// TIA Portal V17 export
// export: Created 2025-03-10T12:18:23.2185831Z, ExportSetting WithDefaults, DisplayName Totally Integrated Automation Portal, DisplayVersion V17 Update 8, DisplayName TIA Portal Openness, DisplayVersion V17 Update 8, DisplayName TIA Portal Version Control Interface, DisplayVersion V17, DisplayName SINAMICS Startdrive Advanced, DisplayVersion V17 SP2, DisplayName SINAMICS Startdrive G110M, G120, G120C, G120D, G120P, G115D, DisplayVersion V17 SP2, DisplayName SINAMICS Startdrive G130, G150, S120, S150, SINAMICS MV, S210, DisplayVersion V17 SP2, DisplayName STEP 7 Professional, DisplayVersion V17 Update 8, DisplayName SINUMERIK ONE STEP 7 Toolbox, DisplayVersion V17 Update 12, DisplayName SINUMERIK 840D sl STEP 7 Toolbox, DisplayVersion V17 Update 12, DisplayName STEP 7 Safety, DisplayVersion V17 Update 6, DisplayName WinCC Advanced, DisplayVersion V17 Update 8
ORGANIZATION_BLOCK "OB1_CYCLE"   // OB1, LAD, ProgramCycle
TITLE = "Main Program Sweep (Cycle)"
{ S7_Optimized_Access := 'FALSE' }
VERSION : 0.1
// stored: AutoNumber false, IsIECCheckEnabled false, SetENOAutomatically false
   VAR_TEMP
      EV_CLASS : Byte;   // Bits 0-3 = 1:Coming event, Bits 4-7 = 1:Event class 1
      SCAN_1 : Byte;   // 1:Initial call of the OB, 3: Call 2-n of the OB
      PRIORITY : Byte;   // Priority of OB Execution
      OB_NUMBR : Byte;   // OB number
      RESERVED_1 : Byte;   // Reserved for system
      RESERVED_2 : Byte;   // Reserved for system
      PREV_CYCLE : Int;   // Previous program cycle time (milliseconds)
      MIN_CYCLE : Int;   // Minimum program cycle time (milliseconds)
      MAX_CYCLE : Int;   // Maximum program cycle time (milliseconds)
      DATE_TIME : Date_And_Time;   // Date and time OB started
      OB1_SCAN : Byte;   // 1 (Cold restart scan 1 of OB 1), 3 (Scan 2-n of OB 1)
      OB1_PRIORITY : Int;   // Priority of OB Execution
      OB1_MIN_CYCLE : DInt;   // Minimum cycle time of OB1 (milliseconds)
      OB1_MAX_CYCLE : DInt;   // Maximum cycle time of OB1 (milliseconds)
      PART_TYPE : Int;
      zero : Byte;
      status_sfc21 : Int;
      Error : Bool;
      status : Word;
   END_VAR
   VAR_TEMP   // added for the SCL form of the ladder/FBD networks
      _w1 : Bool;
   END_VAR
BEGIN

REGION Network 1: M ZERO - M ONE
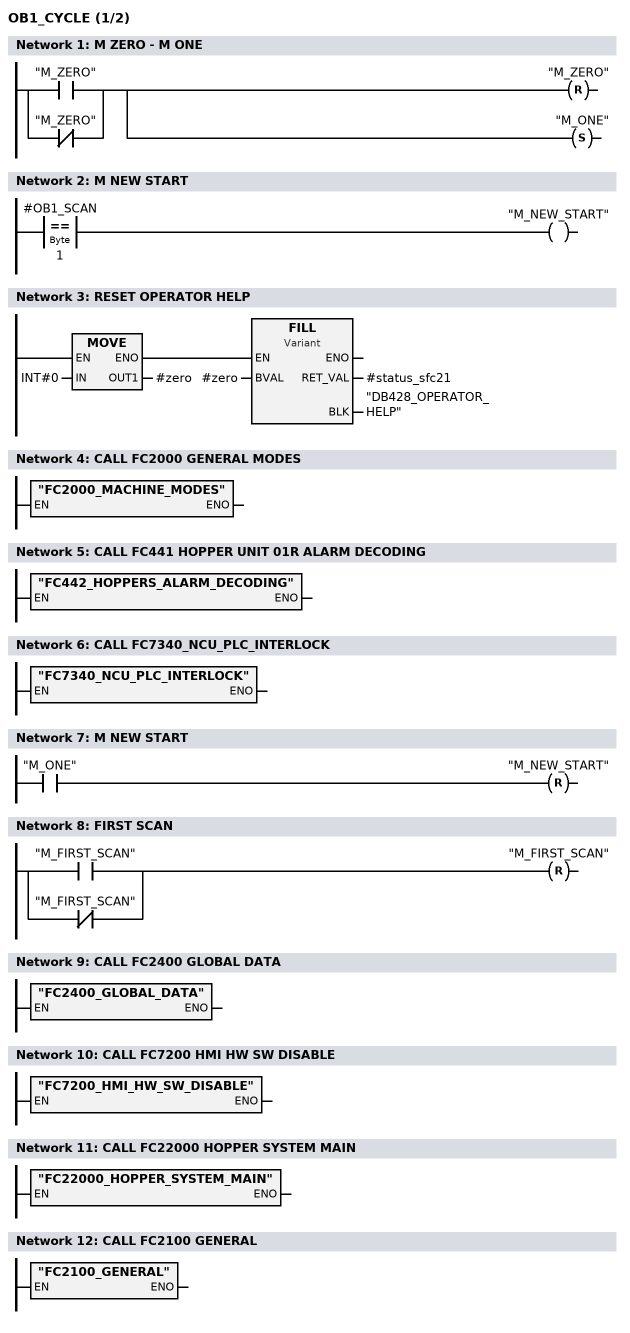
   RUNG wire#powerrail
      Contact( "M_ZERO" )
      wire#w1
      R_Coil( "M_ZERO" )
   END_RUNG
   RUNG wire#powerrail
      I_Contact( "M_ZERO" )
   END_RUNG wire#w1
   RUNG wire#w1
      S_Coil( "M_ONE" )
   END_RUNG
   // the same network as SCL:
   #_w1 := "M_ZERO" OR NOT "M_ZERO";
   IF #_w1 THEN
       "M_ZERO" := FALSE;
       "M_ONE" := TRUE;
   END_IF;
END_REGION

REGION Network 2: M NEW START
   RUNG wire#powerrail
      { S7_Templates := "SrcType := Byte" } EQ_Contact(in1 := #OB1_SCAN, in2 := 1)
      Coil( "M_NEW_START" )
   END_RUNG
   // the same network as SCL:
   "M_NEW_START" := #OB1_SCAN = 1;
END_REGION

REGION Network 3: RESET OPERATOR HELP
   RUNG wire#powerrail
      { S7_GenerateENO := "TRUE" } Move(in := INT#0, out1 => #zero)
      { S7_Templates := "ptr_type := Variant" } FILL(BVAL := #zero, RET_VAL => #status_sfc21, BLK => "DB428_OPERATOR_HELP")
   END_RUNG
   // the same network as SCL:
   // ENO of a box is taken as its EN; it also drops when the box reports an error
   #zero := INT#0;
   #status_sfc21 := FILL(BVAL := #zero, BLK => "DB428_OPERATOR_HELP");
END_REGION

REGION Network 4: CALL FC2000 GENERAL MODES
   RUNG wire#powerrail
      "FC2000_MACHINE_MODES"()
   END_RUNG
   // the same network as SCL:
   "FC2000_MACHINE_MODES"();
END_REGION

REGION Network 5: CALL FC441 HOPPER UNIT 01R ALARM DECODING
   RUNG wire#powerrail
      "FC442_HOPPERS_ALARM_DECODING"()
   END_RUNG
   // the same network as SCL:
   "FC442_HOPPERS_ALARM_DECODING"();
END_REGION

REGION Network 6: CALL FC7340_NCU_PLC_INTERLOCK
   RUNG wire#powerrail
      "FC7340_NCU_PLC_INTERLOCK"()
   END_RUNG
   // the same network as SCL:
   "FC7340_NCU_PLC_INTERLOCK"();
END_REGION

REGION Network 7: M NEW START
   RUNG wire#powerrail
      Contact( "M_ONE" )
      R_Coil( "M_NEW_START" )
   END_RUNG
   // the same network as SCL:
   IF "M_ONE" THEN "M_NEW_START" := FALSE; END_IF;
END_REGION

REGION Network 8: FIRST SCAN
   RUNG wire#powerrail
      Contact( "M_FIRST_SCAN" )
      wire#w1
      R_Coil( "M_FIRST_SCAN" )
   END_RUNG
   RUNG wire#powerrail
      I_Contact( "M_FIRST_SCAN" )
   END_RUNG wire#w1
   // the same network as SCL:
   IF "M_FIRST_SCAN" OR NOT "M_FIRST_SCAN" THEN "M_FIRST_SCAN" := FALSE; END_IF;
END_REGION

REGION Network 9: CALL FC2400 GLOBAL DATA
   RUNG wire#powerrail
      "FC2400_GLOBAL_DATA"()
   END_RUNG
   // the same network as SCL:
   "FC2400_GLOBAL_DATA"();
END_REGION

REGION Network 10: CALL FC7200 HMI HW SW DISABLE
   RUNG wire#powerrail
      "FC7200_HMI_HW_SW_DISABLE"()
   END_RUNG
   // the same network as SCL:
   "FC7200_HMI_HW_SW_DISABLE"();
END_REGION

REGION Network 11: CALL FC22000 HOPPER SYSTEM MAIN
   RUNG wire#powerrail
      "FC22000_HOPPER_SYSTEM_MAIN"()
   END_RUNG
   // the same network as SCL:
   "FC22000_HOPPER_SYSTEM_MAIN"();
END_REGION

REGION Network 12: CALL FC2100 GENERAL
   RUNG wire#powerrail
      "FC2100_GENERAL"()
   END_RUNG
   // the same network as SCL:
   "FC2100_GENERAL"();
END_REGION

REGION Network 13: CALL FC21000 POWDER FEEDER MAIN
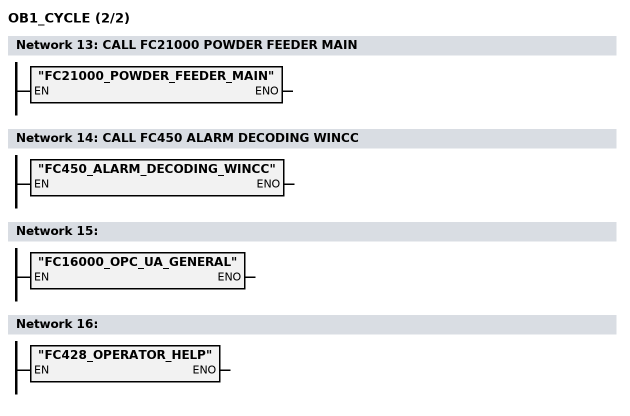
   RUNG wire#powerrail
      "FC21000_POWDER_FEEDER_MAIN"()
   END_RUNG
   // the same network as SCL:
   "FC21000_POWDER_FEEDER_MAIN"();
END_REGION

REGION Network 14: CALL FC450 ALARM DECODING WINCC
   RUNG wire#powerrail
      "FC450_ALARM_DECODING_WINCC"()
   END_RUNG
   // the same network as SCL:
   "FC450_ALARM_DECODING_WINCC"();
END_REGION

REGION Network 15
   RUNG wire#powerrail
      "FC16000_OPC_UA_GENERAL"()
   END_RUNG
   // the same network as SCL:
   "FC16000_OPC_UA_GENERAL"();
END_REGION

REGION Network 16
   RUNG wire#powerrail
      "FC428_OPERATOR_HELP"()
   END_RUNG
   // the same network as SCL:
   "FC428_OPERATOR_HELP"();
END_REGION
END_ORGANIZATION_BLOCK
